Fanuc KAREL source: CA0063.KL

PROGRAM CA0063
%STACKSIZE=65535
%PRIORITY=65535
%NOLOCKGROUP
VAR
G : INTEGER
I : INTEGER
R : REAL
B : BOOLEAN
S : STRING[16]
AI : ARRAY[2] OF INTEGER
AR : ARRAY[2] OF REAL
P : XYZWPR
-- UNRESOLVED DECLARATIONS (source type spelling not recovered)
-- ST : TYPE_0x1100 (type_u16=0x1100)
-- V : TYPE_0x0013 (type_u16=0x0013)
ROUTINE F(P1 : INTEGER; P2 : REAL; P3 : BOOLEAN; P4 : STRING; P5 : ARRAY[*] OF INTEGER; P6 : ARRAY[*] OF REAL; P7 : TYPE_0x1100; P8 : XYZWPR) FROM CA0063
ROUTINE F
BEGIN
G=(G + 1)
END F
BEGIN
G=0
I=1
R=2.5
B=TRUE
S='A'
AI[1]=3
AR[1]=4.5
ST.A=5
ST.B=1087373312
-- UNSAFE_SOURCE_IR line 40: F(ARG_1_UNRESOLVED, ARG_2_UNRESOLVED, ARG_3_UNRESOLVED, ARG_4_UNRESOLVED, ARG_5_UNRESOLVED, ARG_6_UNRESOLVED, ARG_7_UNRESOLVED, ARG_8_UNRESOLVED)
END CA0063
